Staubli VAL3: JogNegative.pgx

public program JogNegative(num x_nAxis, num x_nKey)
begin
  call StepMove(x_nAxis,x_nKey,false)
end
